TYPE ST_BusRelais16F_Cnt_1 :
STRUCT
	dwCntRelais    :ARRAY[1..16] OF DWORD;
END_STRUCT
END_TYPE

(* stored: Version 1.1.0.1, ProductVersion 3.1.4024.12
   DUT ST_BusRelais16F_Cnt_1: Id {cc59452b-caaf-448d-9766-6a78f77743ee} *)
